// TIA Portal project "Dual_Transport_Line" (V19)

(* hardware
DEVICE "S7-1200 station_1"  S7-1200 Station
   slot 0: "Rack_0"  S7-1200 Rack  Rack  V1.0
   slot 1: "PLC_1"  CPU 1215C AC/DC/Rly  6ES7 215-1BG40-0XB0  V4.6
DEVICE "HMI_1"  KTP400 Basic PN
   slot 0: "HMI_1"  KTP400 Basic PN  6AV2 123-2DB03-0AX0  15.1.0.0
   slot 1: "HMI_RT_1"  KTP400 Basic PN  6AV2 123-2DB03-0AX0  15.1.0.0
   slot 5: "HMI_1.IE_CP_1"  PROFINET Interface  15.0.1.0
      slot 1: "PROFINET Interface_1"  PROFINET Interface
         slot 1: "Port_1"  Port
*)

// ===== PLC "PLC_1"  CPU 1215C AC/DC/Rly =====

VAR_GLOBAL   // PLC tag table "Default tag table"
   "System_Byte" AT %MB1 : Byte;
   "FirstScan" AT %M1.0 : Bool;
   "DiagStatusUpdate" AT %M1.1 : Bool;
   "AlwaysTRUE" AT %M1.2 : Bool;
   "AlwaysFALSE" AT %M1.3 : Bool;
   "Clock_Byte" AT %MB0 : Byte;
   "Clock_10Hz" AT %M0.0 : Bool;
   "Clock_5Hz" AT %M0.1 : Bool;
   "Clock_2.5Hz" AT %M0.2 : Bool;
   "Clock_2Hz" AT %M0.3 : Bool;
   "Clock_1.25Hz" AT %M0.4 : Bool;
   "Clock_1Hz" AT %M0.5 : Bool;
   "Clock_0.625Hz" AT %M0.6 : Bool;
   "Clock_0.5Hz" AT %M0.7 : Bool;
END_VAR

VAR_GLOBAL   // PLC tag table "IO"
   "MPCB_01" AT %I0.0 : Bool;   // Motor Protection Circuit Breaker
   "MPCB_02" AT %I0.1 : Bool;   // Motor Protection Circuit Breaker
   "Motor_01" AT %Q0.0 : Bool;
   "Motor_02" AT %Q0.1 : Bool;
END_VAR

TYPE "UDT_Statehandler"
   STRUCT
      State : Struct
         xReady : Bool;
         xRunning : Bool;
         xReset : Bool;
         xFaulted : Bool;
         iState : Int;
      END_STRUCT;
      Command : Struct
         xStart : Bool;
         xStop : Bool;
         xReset : Bool;
      END_STRUCT;
   END_STRUCT;
END_TYPE

TYPE "UDT_Transporter"
   STRUCT
      Status : Struct
         xWith_Package : Bool;
         xFaulted : Bool;
         xRunning : Bool;
         iState : Int;   // 0 - Stop; 10 - Running; 20 - Faulted
      END_STRUCT;
      Command : Struct
         xStart_Sensor : Bool;
         xEnd_Sensor : Bool;
      END_STRUCT;
      Configuration : Struct
         tDowntime : Int;
         iSpeed : Int;
      END_STRUCT;
      Faulted : Struct
         wTrigger : Word;
      END_STRUCT;
   END_STRUCT;
END_TYPE

DATA_BLOCK "Instance - FB - Mirror"   // DB7
{ S7_Optimized_Access := 'TRUE' }
VERSION : 0.1
// stored: InstanceOfName FB - Mirror
"FB - Mirror"
BEGIN
END_DATA_BLOCK

// folder: 00 Machine

DATA_BLOCK "Instance - FB - Statehandler"   // DB2
{ S7_Optimized_Access := 'TRUE' }
VERSION : 0.1
// stored: InstanceOfName FB - Statehandler
"FB - Statehandler"
BEGIN
END_DATA_BLOCK

DATA_BLOCK "Instance - FB - Machine Modules"   // DB3
{ S7_Optimized_Access := 'TRUE' }
VERSION : 0.1
// stored: InstanceOfName FB - Machine Modules
"FB - Machine Modules"
BEGIN
END_DATA_BLOCK

// folder: 01 Equipment/01 Instance

DATA_BLOCK "Instance - FB - Transporter_02"   // DB4
{ S7_Optimized_Access := 'TRUE' }
VERSION : 0.1
// stored: InstanceOfName FB - Transporter
"FB - Transporter"
BEGIN
END_DATA_BLOCK

DATA_BLOCK "Instance - FB - Transporter_01"   // DB6
{ S7_Optimized_Access := 'TRUE' }
VERSION : 0.1
// stored: InstanceOfName FB - Transporter
"FB - Transporter"
BEGIN
END_DATA_BLOCK

DATA_BLOCK "Instance - FB - Equipment Modules"   // DB8
{ S7_Optimized_Access := 'TRUE' }
VERSION : 0.1
// stored: InstanceOfName FB - Equipment Module
"FB - Equipment Module"
BEGIN
END_DATA_BLOCK

DATA_BLOCK "Instance - FB - Package_Position"   // DB9
{ S7_Optimized_Access := 'TRUE' }
VERSION : 0.1
// stored: InstanceOfName FB - Package_Position
"FB - Package_Position"
BEGIN
END_DATA_BLOCK

DATA_BLOCK "Instance - FB - Sensor_01"   // DB10
{ S7_Optimized_Access := 'TRUE' }
VERSION : 0.1
// stored: InstanceOfName FB - Sensor
"FB - Sensor"
BEGIN
END_DATA_BLOCK

DATA_BLOCK "Instance - FB - Sensor_02"   // DB11
{ S7_Optimized_Access := 'TRUE' }
VERSION : 0.1
// stored: InstanceOfName FB - Sensor
"FB - Sensor"
BEGIN
END_DATA_BLOCK

DATA_BLOCK "Instance - Package_Counter"   // DB12
{ S7_Optimized_Access := 'TRUE' }
VERSION : 0.1
// stored: InstanceOfName Package_Counter
"Package_Counter"
BEGIN
END_DATA_BLOCK

// folder: 02 Global Data

DATA_BLOCK "DB - Statehandler"   // DB1
{ S7_Optimized_Access := 'TRUE' }
VERSION : 0.1
   VAR
      Statehandler : "UDT_Statehandler";
   END_VAR
BEGIN
END_DATA_BLOCK

DATA_BLOCK "DB - Equipment"   // DB5
{ S7_Optimized_Access := 'TRUE' }
VERSION : 0.1
   VAR
      Transporter_01 : "UDT_Transporter";
      Transporter_02 : "UDT_Transporter";
      iPackage_Position : Int;
      iPackage_Count : Int;
   END_VAR
BEGIN
END_DATA_BLOCK

// folder: (top level)

FUNCTION_BLOCK "FB - Mirror"   // FB3, LAD
{ S7_Optimized_Access := 'TRUE' }
VERSION : 0.1
BEGIN

REGION Network 1: Motor Protection Circuit Breaker
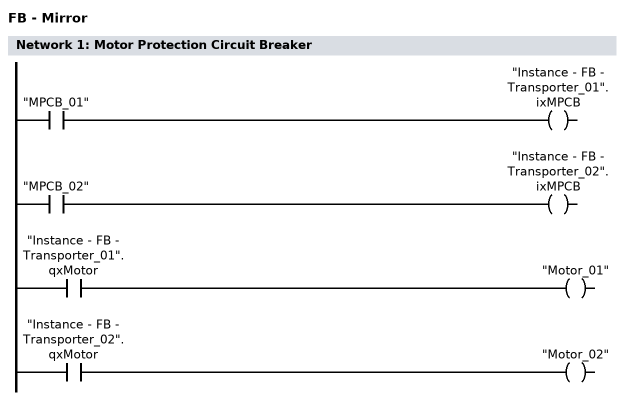
   RUNG wire#powerrail
      Contact( "MPCB_01" )
      Coil( "Instance - FB - Transporter_01".ixMPCB )
   END_RUNG
   RUNG wire#powerrail
      Contact( "MPCB_02" )
      Coil( "Instance - FB - Transporter_02".ixMPCB )
   END_RUNG
   RUNG wire#powerrail
      Contact( "Instance - FB - Transporter_01".qxMotor )
      Coil( "Motor_01" )
   END_RUNG
   RUNG wire#powerrail
      Contact( "Instance - FB - Transporter_02".qxMotor )
      Coil( "Motor_02" )
   END_RUNG
   // the same network as SCL:
   "Instance - FB - Transporter_01".ixMPCB := "MPCB_01";
   "Instance - FB - Transporter_02".ixMPCB := "MPCB_02";
   "Motor_01" := "Instance - FB - Transporter_01".qxMotor;
   "Motor_02" := "Instance - FB - Transporter_02".qxMotor;
END_REGION
END_FUNCTION_BLOCK

ORGANIZATION_BLOCK "Main"   // OB1, LAD, ProgramCycle
TITLE = "Main Program Sweep (Cycle)"
{ S7_Optimized_Access := 'TRUE' }
VERSION : 0.1
   VAR_INPUT
      Initial_Call : Bool;   // Initial call of this OB
      Remanence : Bool;   // =True, if remanent data are available
   END_VAR
BEGIN

REGION Network 1: CALL MACHINE MODULES
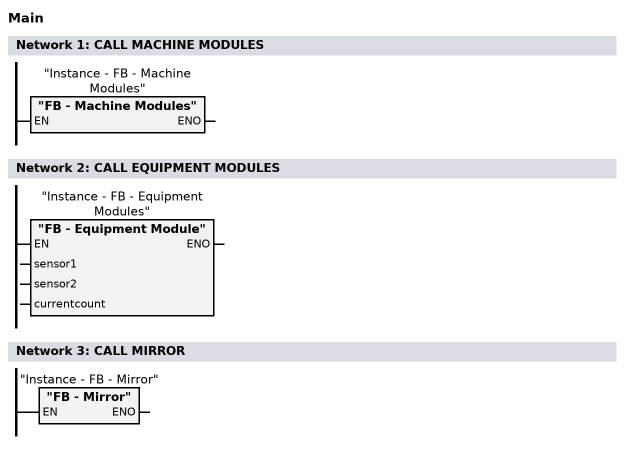
   RUNG wire#powerrail
      "Instance - FB - Machine Modules"()
   END_RUNG
   // the same network as SCL:
   "Instance - FB - Machine Modules"();   // "FB - Machine Modules"
END_REGION

REGION Network 2: CALL EQUIPMENT MODULES
   RUNG wire#powerrail
      "Instance - FB - Equipment Modules"(sensor1 :=, sensor2 :=, currentcount :=)
   END_RUNG
   // the same network as SCL:
   "Instance - FB - Equipment Modules"();   // "FB - Equipment Module"
END_REGION

REGION Network 3: CALL MIRROR
   RUNG wire#powerrail
      "Instance - FB - Mirror"()
   END_RUNG
   // the same network as SCL:
   "Instance - FB - Mirror"();   // "FB - Mirror"
END_REGION
END_ORGANIZATION_BLOCK

// folder: 00 Machine

FUNCTION_BLOCK "FB - Statehandler"   // FB1, LAD
{ S7_Optimized_Access := 'TRUE' }
VERSION : 0.1
   VAR_INPUT
      Transporter_01 : "UDT_Transporter";
      Transporter_02 : "UDT_Transporter";
   END_VAR
   VAR_IN_OUT
      "DB Statehandler" : "UDT_Statehandler";
   END_VAR
   VAR
      "xActive Faulted" : Bool;
      R_TRIG_Start : R_TRIG;
      R_TRIG_Stop : R_TRIG;
      R_TRIG_Reset : R_TRIG;
      xGlobal_Faulted : Bool;
   END_VAR
BEGIN

REGION Network 1: GLOBAL FAULTED
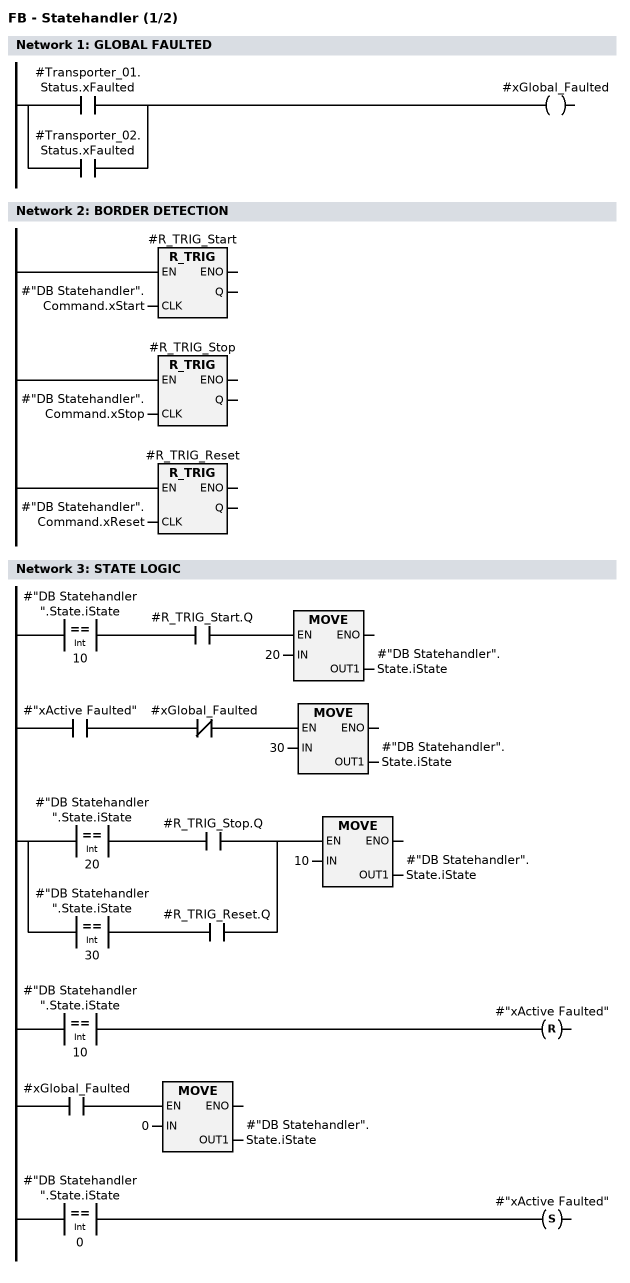
   RUNG wire#powerrail
      Contact( #Transporter_01.Status.xFaulted )
      wire#w1
      Coil( #xGlobal_Faulted )
   END_RUNG
   RUNG wire#powerrail
      Contact( #Transporter_02.Status.xFaulted )
   END_RUNG wire#w1
   // the same network as SCL:
   #xGlobal_Faulted := #Transporter_01.Status.xFaulted OR #Transporter_02.Status.xFaulted;
END_REGION

REGION Network 2: BORDER DETECTION
   #R_TRIG_Start(CLK := #"DB Statehandler".Command.xStart);   // R_TRIG
   #R_TRIG_Stop(CLK := #"DB Statehandler".Command.xStop);   // R_TRIG
   #R_TRIG_Reset(CLK := #"DB Statehandler".Command.xReset);   // R_TRIG
END_REGION

REGION Network 3: STATE LOGIC
   RUNG wire#powerrail
      { S7_Templates := "SrcType := Int" } EQ_Contact(in1 := #"DB Statehandler".State.iState, in2 := 10)
      Contact( #R_TRIG_Start.Q )
      Move(in := 20, out1 => #"DB Statehandler".State.iState)
   END_RUNG
   RUNG wire#powerrail
      Contact( #"xActive Faulted" )
      I_Contact( #xGlobal_Faulted )
      Move(in := 30, out1 => #"DB Statehandler".State.iState)
   END_RUNG
   RUNG wire#powerrail
      { S7_Templates := "SrcType := Int" } EQ_Contact(in1 := #"DB Statehandler".State.iState, in2 := 20)
      Contact( #R_TRIG_Stop.Q )
      wire#w1
      Move(in := 10, out1 => #"DB Statehandler".State.iState)
   END_RUNG
   RUNG wire#powerrail
      { S7_Templates := "SrcType := Int" } EQ_Contact(in1 := #"DB Statehandler".State.iState, in2 := 30)
      Contact( #R_TRIG_Reset.Q )
   END_RUNG wire#w1
   RUNG wire#powerrail
      { S7_Templates := "SrcType := Int" } EQ_Contact(in1 := #"DB Statehandler".State.iState, in2 := 10)
      R_Coil( #"xActive Faulted" )
   END_RUNG
   RUNG wire#powerrail
      Contact( #xGlobal_Faulted )
      Move(in := 0, out1 => #"DB Statehandler".State.iState)
   END_RUNG
   RUNG wire#powerrail
      { S7_Templates := "SrcType := Int" } EQ_Contact(in1 := #"DB Statehandler".State.iState, in2 := 0)
      S_Coil( #"xActive Faulted" )
   END_RUNG
   // the same network as SCL:
   IF (#"DB Statehandler".State.iState = 10) AND #R_TRIG_Start.Q THEN
       #"DB Statehandler".State.iState := 20;
   END_IF;
   IF #"xActive Faulted" AND NOT #xGlobal_Faulted THEN #"DB Statehandler".State.iState := 30; END_IF;
   IF ((#"DB Statehandler".State.iState = 20) AND #R_TRIG_Stop.Q) OR ((#"DB Statehandler".State.iState = 30) AND #R_TRIG_Reset.Q) THEN
       #"DB Statehandler".State.iState := 10;
   END_IF;
   IF #"DB Statehandler".State.iState = 10 THEN #"xActive Faulted" := FALSE; END_IF;
   IF #xGlobal_Faulted THEN #"DB Statehandler".State.iState := 0; END_IF;
   IF #"DB Statehandler".State.iState = 0 THEN #"xActive Faulted" := TRUE; END_IF;
END_REGION

REGION Network 4: TRIGGERS
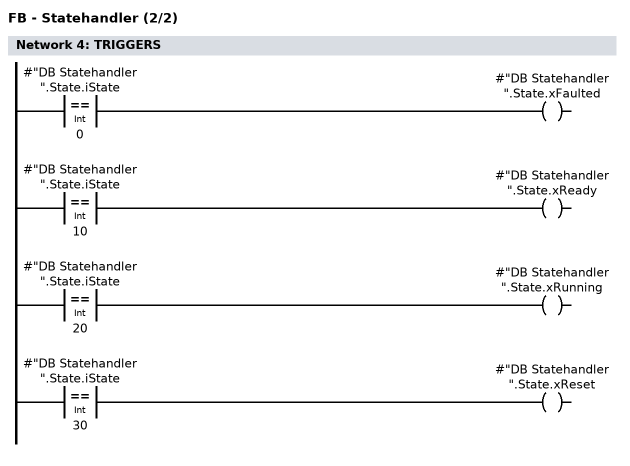
   RUNG wire#powerrail
      { S7_Templates := "SrcType := Int" } EQ_Contact(in1 := #"DB Statehandler".State.iState, in2 := 0)
      Coil( #"DB Statehandler".State.xFaulted )
   END_RUNG
   RUNG wire#powerrail
      { S7_Templates := "SrcType := Int" } EQ_Contact(in1 := #"DB Statehandler".State.iState, in2 := 10)
      Coil( #"DB Statehandler".State.xReady )
   END_RUNG
   RUNG wire#powerrail
      { S7_Templates := "SrcType := Int" } EQ_Contact(in1 := #"DB Statehandler".State.iState, in2 := 20)
      Coil( #"DB Statehandler".State.xRunning )
   END_RUNG
   RUNG wire#powerrail
      { S7_Templates := "SrcType := Int" } EQ_Contact(in1 := #"DB Statehandler".State.iState, in2 := 30)
      Coil( #"DB Statehandler".State.xReset )
   END_RUNG
   // the same network as SCL:
   #"DB Statehandler".State.xFaulted := #"DB Statehandler".State.iState = 0;
   #"DB Statehandler".State.xReady := #"DB Statehandler".State.iState = 10;
   #"DB Statehandler".State.xRunning := #"DB Statehandler".State.iState = 20;
   #"DB Statehandler".State.xReset := #"DB Statehandler".State.iState = 30;
END_REGION
END_FUNCTION_BLOCK

FUNCTION_BLOCK "FB - Machine Modules"   // FB2, LAD
{ S7_Optimized_Access := 'TRUE' }
VERSION : 0.1
BEGIN

REGION Network 1
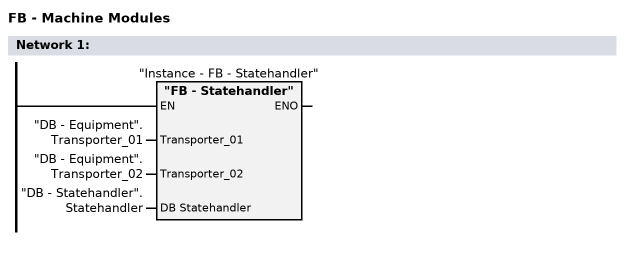
   RUNG wire#powerrail
      "Instance - FB - Statehandler"(Transporter_01 := "DB - Equipment".Transporter_01, Transporter_02 := "DB - Equipment".Transporter_02, "DB Statehandler" := "DB - Statehandler".Statehandler)
   END_RUNG
   // the same network as SCL:
   "Instance - FB - Statehandler"(Transporter_01 := "DB - Equipment".Transporter_01,   // "FB - Statehandler"
                           Transporter_02 := "DB - Equipment".Transporter_02,
                           "DB Statehandler" := "DB - Statehandler".Statehandler);
END_REGION
END_FUNCTION_BLOCK

// folder: 01 Equipment/00 Function

FUNCTION_BLOCK "FB - Equipment Module"   // FB4, LAD
{ S7_Optimized_Access := 'TRUE' }
VERSION : 0.1
   VAR_INPUT
      sensor1 : Bool;
      sensor2 : Bool;
      currentcount : DInt;
   END_VAR
BEGIN

REGION Network 1: CALL TRANSPORTER
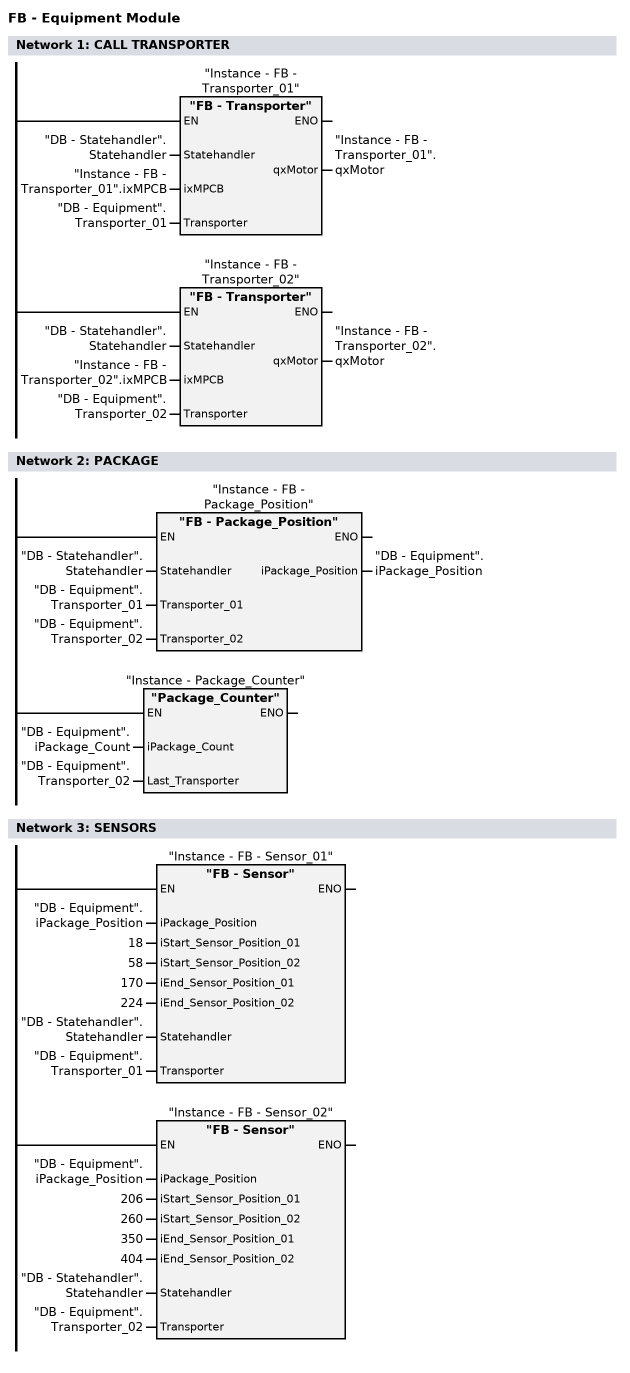
   RUNG wire#powerrail
      "Instance - FB - Transporter_01"(Statehandler := "DB - Statehandler".Statehandler, ixMPCB := "Instance - FB - Transporter_01".ixMPCB, Transporter := "DB - Equipment".Transporter_01, qxMotor => "Instance - FB - Transporter_01".qxMotor)
   END_RUNG
   RUNG wire#powerrail
      "Instance - FB - Transporter_02"(Statehandler := "DB - Statehandler".Statehandler, ixMPCB := "Instance - FB - Transporter_02".ixMPCB, Transporter := "DB - Equipment".Transporter_02, qxMotor => "Instance - FB - Transporter_02".qxMotor)
   END_RUNG
   // the same network as SCL:
   "Instance - FB - Transporter_01"(Statehandler := "DB - Statehandler".Statehandler,   // "FB - Transporter"
                           ixMPCB := "Instance - FB - Transporter_01".ixMPCB,
                           Transporter := "DB - Equipment".Transporter_01,
                           qxMotor => "Instance - FB - Transporter_01".qxMotor);
   "Instance - FB - Transporter_02"(Statehandler := "DB - Statehandler".Statehandler,   // "FB - Transporter"
                           ixMPCB := "Instance - FB - Transporter_02".ixMPCB,
                           Transporter := "DB - Equipment".Transporter_02,
                           qxMotor => "Instance - FB - Transporter_02".qxMotor);
END_REGION

REGION Network 2: PACKAGE
   RUNG wire#powerrail
      "Instance - FB - Package_Position"(Statehandler := "DB - Statehandler".Statehandler, Transporter_01 := "DB - Equipment".Transporter_01, Transporter_02 := "DB - Equipment".Transporter_02, iPackage_Position => "DB - Equipment".iPackage_Position)
   END_RUNG
   RUNG wire#powerrail
      "Instance - Package_Counter"(iPackage_Count := "DB - Equipment".iPackage_Count, Last_Transporter := "DB - Equipment".Transporter_02)
   END_RUNG
   // the same network as SCL:
   "Instance - FB - Package_Position"(Statehandler := "DB - Statehandler".Statehandler,   // "FB - Package_Position"
                           Transporter_01 := "DB - Equipment".Transporter_01,
                           Transporter_02 := "DB - Equipment".Transporter_02,
                           iPackage_Position => "DB - Equipment".iPackage_Position);
   "Instance - Package_Counter"(iPackage_Count := "DB - Equipment".iPackage_Count,   // "Package_Counter"
                           Last_Transporter := "DB - Equipment".Transporter_02);
END_REGION

REGION Network 3: SENSORS
   RUNG wire#powerrail
      "Instance - FB - Sensor_01"(iPackage_Position := "DB - Equipment".iPackage_Position, iStart_Sensor_Position_01 := 18, iStart_Sensor_Position_02 := 58, iEnd_Sensor_Position_01 := 170, iEnd_Sensor_Position_02 := 224, Statehandler := "DB - Statehandler".Statehandler, Transporter := "DB - Equipment".Transporter_01)
   END_RUNG
   RUNG wire#powerrail
      "Instance - FB - Sensor_02"(iPackage_Position := "DB - Equipment".iPackage_Position, iStart_Sensor_Position_01 := 206, iStart_Sensor_Position_02 := 260, iEnd_Sensor_Position_01 := 350, iEnd_Sensor_Position_02 := 404, Statehandler := "DB - Statehandler".Statehandler, Transporter := "DB - Equipment".Transporter_02)
   END_RUNG
   // the same network as SCL:
   "Instance - FB - Sensor_01"(iPackage_Position := "DB - Equipment".iPackage_Position,   // "FB - Sensor"
                           iStart_Sensor_Position_01 := 18,
                           iStart_Sensor_Position_02 := 58,
                           iEnd_Sensor_Position_01 := 170,
                           iEnd_Sensor_Position_02 := 224,
                           Statehandler := "DB - Statehandler".Statehandler,
                           Transporter := "DB - Equipment".Transporter_01);
   "Instance - FB - Sensor_02"(iPackage_Position := "DB - Equipment".iPackage_Position,   // "FB - Sensor"
                           iStart_Sensor_Position_01 := 206,
                           iStart_Sensor_Position_02 := 260,
                           iEnd_Sensor_Position_01 := 350,
                           iEnd_Sensor_Position_02 := 404,
                           Statehandler := "DB - Statehandler".Statehandler,
                           Transporter := "DB - Equipment".Transporter_02);
END_REGION
END_FUNCTION_BLOCK

FUNCTION_BLOCK "FB - Transporter"   // FB5, LAD
{ S7_Optimized_Access := 'TRUE' }
VERSION : 0.1
   VAR_INPUT
      Statehandler : "UDT_Statehandler";
      ixMPCB : Bool;   // Motor Protection Circuit Breaker
   END_VAR
   VAR_OUTPUT
      qxMotor : Bool;
   END_VAR
   VAR_IN_OUT
      Transporter : "UDT_Transporter";
   END_VAR
   VAR
      F_TRIG_Sensor_End : F_TRIG;
      TOF_Downtime : TOF_TIME;
      iDowntime_MS : DInt;
   END_VAR
BEGIN

REGION Network 1: CONVERT UNITS
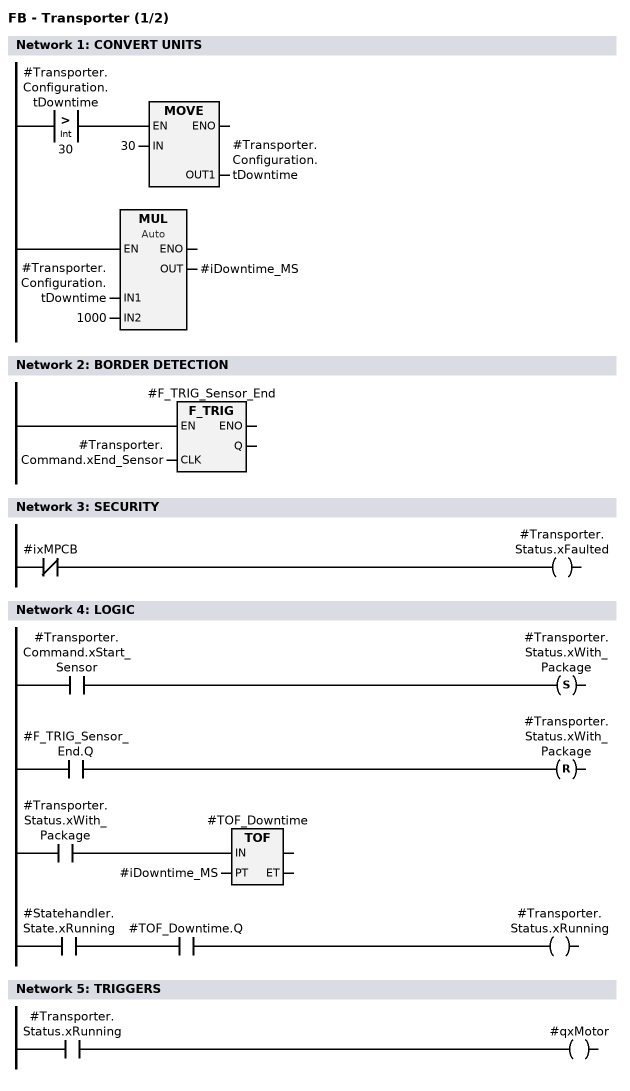
   RUNG wire#powerrail
      { S7_Templates := "SrcType := Int" } GT_Contact(in1 := #Transporter.Configuration.tDowntime, in2 := 30)
      Move(in := 30, out1 => #Transporter.Configuration.tDowntime)
   END_RUNG
   RUNG wire#powerrail
      Mul(in1 := #Transporter.Configuration.tDowntime, in2 := 1000, out => #iDowntime_MS)
   END_RUNG
   // the same network as SCL:
   IF #Transporter.Configuration.tDowntime > 30 THEN #Transporter.Configuration.tDowntime := 30; END_IF;
   #iDowntime_MS := #Transporter.Configuration.tDowntime * 1000;
END_REGION

REGION Network 2: BORDER DETECTION
   #F_TRIG_Sensor_End(CLK := #Transporter.Command.xEnd_Sensor);   // F_TRIG
END_REGION

REGION Network 3: SECURITY
   RUNG wire#powerrail
      I_Contact( #ixMPCB )
      Coil( #Transporter.Status.xFaulted )
   END_RUNG
   // the same network as SCL:
   #Transporter.Status.xFaulted := NOT #ixMPCB;
END_REGION

REGION Network 4: LOGIC
   IF #Transporter.Command.xStart_Sensor THEN #Transporter.Status.xWith_Package := TRUE; END_IF;
   IF #F_TRIG_Sensor_End.Q THEN #Transporter.Status.xWith_Package := FALSE; END_IF;
   #TOF_Downtime(IN := #Transporter.Status.xWith_Package, PT := #iDowntime_MS);   // TOF
   #Transporter.Status.xRunning := #Statehandler.State.xRunning AND #TOF_Downtime.Q;
END_REGION

REGION Network 5: TRIGGERS
   RUNG wire#powerrail
      Contact( #Transporter.Status.xRunning )
      Coil( #qxMotor )
   END_RUNG
   // the same network as SCL:
   #qxMotor := #Transporter.Status.xRunning;
END_REGION

REGION Network 6: STATUS
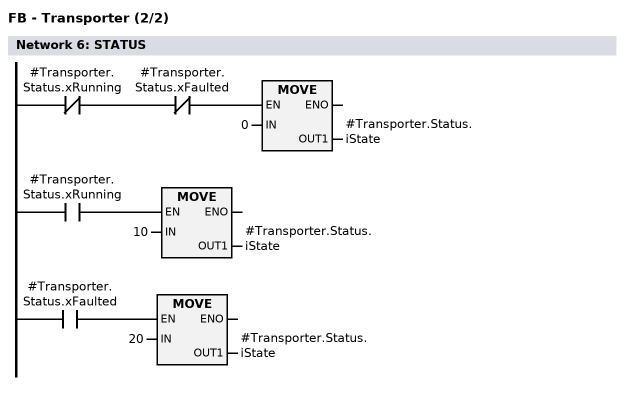
   RUNG wire#powerrail
      I_Contact( #Transporter.Status.xRunning )
      I_Contact( #Transporter.Status.xFaulted )
      Move(in := 0, out1 => #Transporter.Status.iState)
   END_RUNG
   RUNG wire#powerrail
      Contact( #Transporter.Status.xRunning )
      Move(in := 10, out1 => #Transporter.Status.iState)
   END_RUNG
   RUNG wire#powerrail
      Contact( #Transporter.Status.xFaulted )
      Move(in := 20, out1 => #Transporter.Status.iState)
   END_RUNG
   // the same network as SCL:
   IF NOT #Transporter.Status.xRunning AND NOT #Transporter.Status.xFaulted THEN
       #Transporter.Status.iState := 0;
   END_IF;
   IF #Transporter.Status.xRunning THEN #Transporter.Status.iState := 10; END_IF;
   IF #Transporter.Status.xFaulted THEN #Transporter.Status.iState := 20; END_IF;
END_REGION
END_FUNCTION_BLOCK

FUNCTION_BLOCK "FB - Package_Position"   // FB6, LAD
{ S7_Optimized_Access := 'TRUE' }
VERSION : 0.1
   VAR_OUTPUT
      iPackage_Position : Int := 36;
   END_VAR
   VAR_IN_OUT
      Statehandler : "UDT_Statehandler";
      Transporter_01 : "UDT_Transporter";
      Transporter_02 : "UDT_Transporter";
   END_VAR
   VAR
      R_TRIG_Clock : R_TRIG;
      "Instance - FB - Clock_Transporter_01" : "FB - Clock";
      "Instance - FB - Clock_Transporter_02" : "FB - Clock";
      rRPM_Norm_Transporter_02 : Real;
      iTime_Before_Convert_01 : Int;
      iTime_Before_Convert_02 : DInt;
      tTime_Transporter_01 : Time;
      tTime_Transporter_02 : Time;
   END_VAR
BEGIN

REGION Network 1: CLOCK
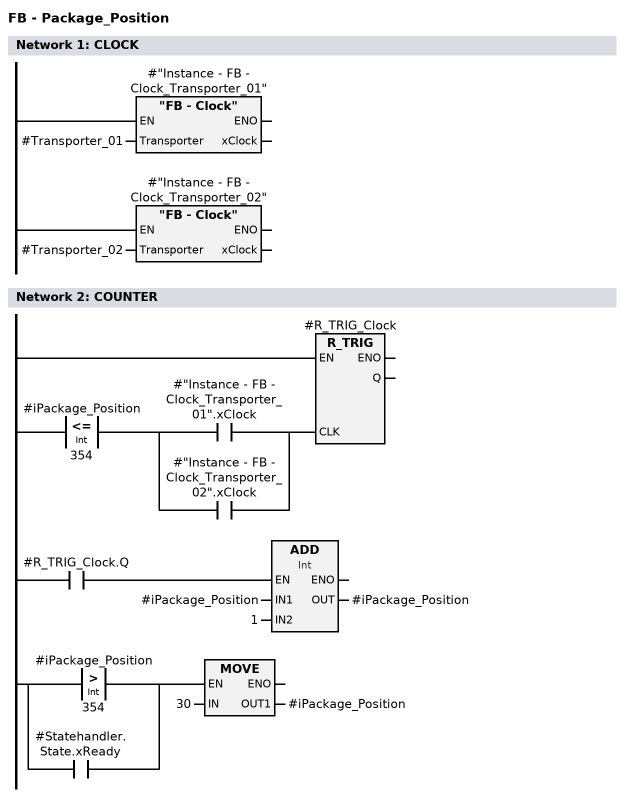
   RUNG wire#powerrail
      #"Instance - FB - Clock_Transporter_01"(Transporter := #Transporter_01, xClock =>)
   END_RUNG
   RUNG wire#powerrail
      #"Instance - FB - Clock_Transporter_02"(Transporter := #Transporter_02, xClock =>)
   END_RUNG
   // the same network as SCL:
   #"Instance - FB - Clock_Transporter_01"(Transporter := #Transporter_01);   // "FB - Clock"
   #"Instance - FB - Clock_Transporter_02"(Transporter := #Transporter_02);   // "FB - Clock"
END_REGION

REGION Network 2: COUNTER
   #R_TRIG_Clock(CLK := (#iPackage_Position <= 354) AND (#"Instance - FB - Clock_Transporter_01".xClock OR #"Instance - FB - Clock_Transporter_02".xClock));   // R_TRIG
   IF #R_TRIG_Clock.Q THEN #iPackage_Position := #iPackage_Position + 1; END_IF;
   IF (#iPackage_Position > 354) OR #Statehandler.State.xReady THEN #iPackage_Position := 30; END_IF;
END_REGION
END_FUNCTION_BLOCK

FUNCTION_BLOCK "FB - Sensor"   // FB7, LAD
{ S7_Optimized_Access := 'TRUE' }
VERSION : 0.1
   VAR_INPUT
      iPackage_Position : Int;
      iStart_Sensor_Position_01 : Int;
      iStart_Sensor_Position_02 : Int;
      iEnd_Sensor_Position_01 : Int;
      iEnd_Sensor_Position_02 : Int;
   END_VAR
   VAR_IN_OUT
      Statehandler : "UDT_Statehandler";
      Transporter : "UDT_Transporter";
   END_VAR
BEGIN

REGION Network 1
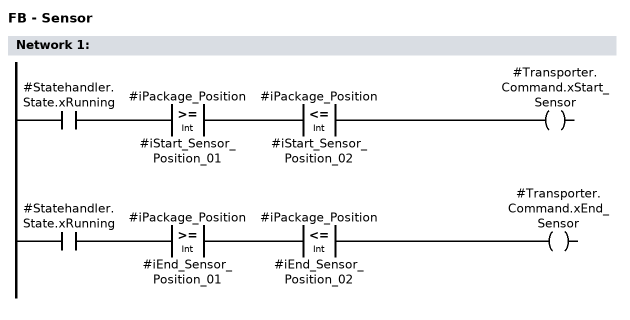
   RUNG wire#powerrail
      Contact( #Statehandler.State.xRunning )
      { S7_Templates := "SrcType := Int" } GE_Contact(in1 := #iPackage_Position, in2 := #iStart_Sensor_Position_01)
      { S7_Templates := "SrcType := Int" } LE_Contact(in1 := #iPackage_Position, in2 := #iStart_Sensor_Position_02)
      Coil( #Transporter.Command.xStart_Sensor )
   END_RUNG
   RUNG wire#powerrail
      Contact( #Statehandler.State.xRunning )
      { S7_Templates := "SrcType := Int" } GE_Contact(in1 := #iPackage_Position, in2 := #iEnd_Sensor_Position_01)
      { S7_Templates := "SrcType := Int" } LE_Contact(in1 := #iPackage_Position, in2 := #iEnd_Sensor_Position_02)
      Coil( #Transporter.Command.xEnd_Sensor )
   END_RUNG
   // the same network as SCL:
   #Transporter.Command.xStart_Sensor := #Statehandler.State.xRunning AND (#iPackage_Position >= #iStart_Sensor_Position_01) AND (#iPackage_Position <= #iStart_Sensor_Position_02);
   #Transporter.Command.xEnd_Sensor := #Statehandler.State.xRunning AND (#iPackage_Position >= #iEnd_Sensor_Position_01) AND (#iPackage_Position <= #iEnd_Sensor_Position_02);
END_REGION
END_FUNCTION_BLOCK

FUNCTION_BLOCK "Package_Counter"   // FB8, LAD
{ S7_Optimized_Access := 'TRUE' }
VERSION : 0.1
   VAR_IN_OUT
      iPackage_Count : Int;
      Last_Transporter : "UDT_Transporter";
   END_VAR
   VAR RETAIN
      "Counter" : CTU_INT;
   END_VAR
BEGIN

REGION Network 1
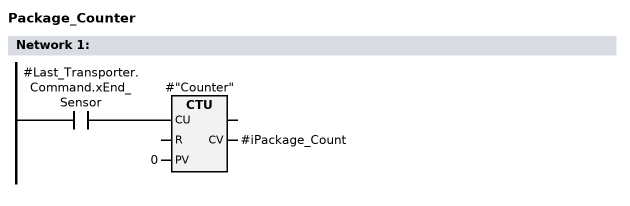
   #"Counter"(CU := #Last_Transporter.Command.xEnd_Sensor, PV := 0, CV => #iPackage_Count);   // CTU
END_REGION
END_FUNCTION_BLOCK

FUNCTION_BLOCK "FB - Clock"   // FB9, LAD
{ S7_Optimized_Access := 'TRUE' }
VERSION : 0.1
   VAR_OUTPUT
      xClock : Bool;
   END_VAR
   VAR_IN_OUT
      Transporter : "UDT_Transporter";
   END_VAR
   VAR
      TON_01 : TON_TIME;
      TON_02 : TON_TIME;
      rSpeed_Convert : Real;
      rTIme_Calculated : Real;
      iTime_Calculated : DInt;
      tTIme : Time;
   END_VAR
BEGIN

REGION Network 1: SPEED LIMIT
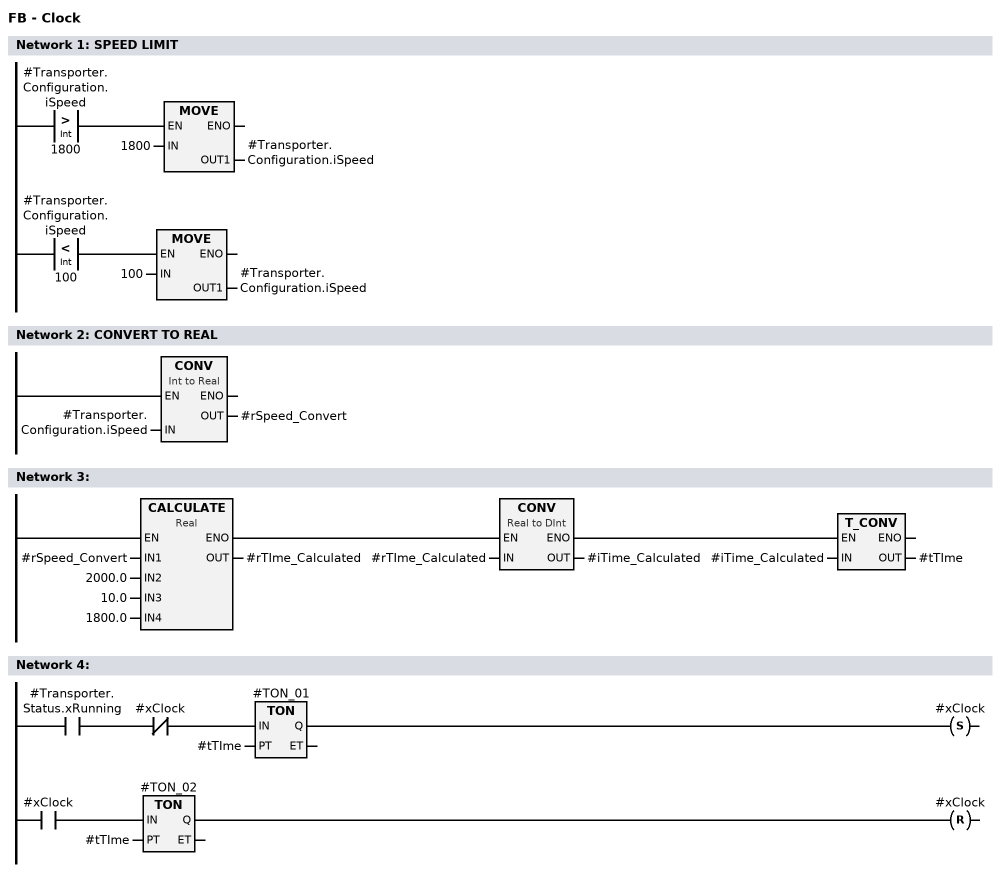
   RUNG wire#powerrail
      { S7_Templates := "SrcType := Int" } GT_Contact(in1 := #Transporter.Configuration.iSpeed, in2 := 1800)
      Move(in := 1800, out1 => #Transporter.Configuration.iSpeed)
   END_RUNG
   RUNG wire#powerrail
      { S7_Templates := "SrcType := Int" } LT_Contact(in1 := #Transporter.Configuration.iSpeed, in2 := 100)
      Move(in := 100, out1 => #Transporter.Configuration.iSpeed)
   END_RUNG
   // the same network as SCL:
   IF #Transporter.Configuration.iSpeed > 1800 THEN #Transporter.Configuration.iSpeed := 1800; END_IF;
   IF #Transporter.Configuration.iSpeed < 100 THEN #Transporter.Configuration.iSpeed := 100; END_IF;
END_REGION

REGION Network 2: CONVERT TO REAL
   RUNG wire#powerrail
      { S7_Templates := "[SrcType := Int, DestType := Real]" } Convert(in := #Transporter.Configuration.iSpeed, out => #rSpeed_Convert)
   END_RUNG
   // the same network as SCL:
   #rSpeed_Convert := INT_TO_REAL(#Transporter.Configuration.iSpeed);
END_REGION

REGION Network 3
   #rTIme_Calculated := 2000.0 - ((#rSpeed_Convert / 1800.0) * (2000.0 -  10.0));
   #iTime_Calculated := REAL_TO_DINT(#rTIme_Calculated);
   #tTIme := T_CONV(IN := #iTime_Calculated);
END_REGION

REGION Network 4
   #TON_01(IN := #Transporter.Status.xRunning AND NOT #xClock, PT := #tTIme);   // TON
   IF #TON_01.Q THEN #xClock := TRUE; END_IF;
   #TON_02(IN := #xClock, PT := #tTIme);   // TON
   IF #TON_02.Q THEN #xClock := FALSE; END_IF;
END_REGION
END_FUNCTION_BLOCK

(* ===== HMI "HMI_RT_1" =====
system functions are stored by id; their names below are inferred from use
connection "HMI_Connection_1": ETHERNET, SMART_S7_1200_OMS

HMI tags "Login Tags"
   "_iScreenNumber" : Int, internal
   "_iUsername_Group" : Int, internal
   "_sUsername" : WString[254], internal
   "_sInputUsername" : WString[254], internal
   "_sInputPassword" : WString[254], internal

HMI tags "Template Command Tags"
   "_xState_Btn_Alarm" : Bool, internal
   "_xState_Btn_Overview" : Bool, internal
   "_xState_Btn_Recipes" : Bool, internal
   "_xState_Btn_Settings" : Bool, internal

HMI tags "Configuration Tags"
   "DB - Equipment_Transporter_01_Configuration_iSpeed" : Int = PLC "DB - Equipment".Transporter_01.Configuration.iSpeed, 100 ms
   "DB - Equipment_Transporter_01_Configuration_tDowntime" : Int = PLC "DB - Equipment".Transporter_01.Configuration.tDowntime, 100 ms
   "DB - Equipment_Transporter_02_Configuration_iSpeed" : Int = PLC "DB - Equipment".Transporter_02.Configuration.iSpeed, 100 ms
   "DB - Equipment_Transporter_02_Configuration_tDowntime" : Int = PLC "DB - Equipment".Transporter_02.Configuration.tDowntime, 100 ms

HMI tags "Status Tags"
   "DB - Equipment_iPackage_Count" : Int = PLC "DB - Equipment".iPackage_Count, 100 ms
   "DB - Equipment_iPackage_Position" : Int = PLC "DB - Equipment".iPackage_Position, 100 ms
   "DB - Equipment_Transporter_01_Faulted_wTrigger" : Word = PLC "DB - Equipment".Transporter_01.Faulted.wTrigger, 1 s
   "DB - Equipment_Transporter_01_Status_iState" : Int = PLC "DB - Equipment".Transporter_01.Status.iState, 100 ms
   "DB - Equipment_Transporter_02_Faulted_wTrigger" : Word = PLC "DB - Equipment".Transporter_02.Faulted.wTrigger, 1 s
   "DB - Equipment_Transporter_02_Status_iState" : Int = PLC "DB - Equipment".Transporter_02.Status.iState, 100 ms
   "DB - Statehandler_Statehandler" : UDT_Statehandler = PLC "DB - Statehandler".Statehandler AT %DB1.DBX0.0, 100 ms

analog alarms
   1: 'Fault detected in Transporter 01', class Errors, trigger "DB - Equipment_Transporter_01_Status_iState"
   2: 'Fault detected in Transporter 02', class Errors, trigger "DB - Equipment_Transporter_02_Status_iState"

graphic list "GraphicList_Btn_template_Overview": 0 'Btn_Template_Overview_Off'; 1 'Btn_Template_Overview_On'

graphic list "GraphicList_Btn_template_Alarm": 0 'Btn_Template_Alert_Off'; 1 'Btn_Template_Alert_On'

graphic list "GraphicList_Btn_template_Recipes": 0 'Btn_Template_Recipe_Off'; 1 'Btn_Template_Recipe_On'

graphic list "GraphicList_Btn_template_Settings": 0 'Btn_Template_Settings_Off'; 1 'Btn_Template_Settings_On'

graphic list "GraphicList_Motor_01": 0 'Graphic_7'; 10 'Graphic_8'; 20 'Graphic_9'

recipe "Product A": Speed_Motor_01 <- "DB - Equipment_Transporter_01_Configuration_iSpeed", Speed_Motor_02 <- "DB - Equipment_Transporter_02_Configuration_iSpeed", Downtime_Motor_01 <- "DB - Equipment_Transporter_01_Configuration_tDowntime", Downtime_Motor_02 <- "DB - Equipment_Transporter_02_Configuration_tDowntime"

Template "Template" 480x272
   Rectangle "Template_Rectangle_4" at 4,24 size 427x242
      Appearance <- "iState"
   Button "Template_Button_1" at 435,0 size 45x45; TextOff 'Text'; PictureList "GraphicList_Btn_template_Overview"
      ProcessValue <- "_xState_Btn_Overview"
      on Release: ActivateScreen("1 OVERVIEW", 0)
   Button "Template_Button_2" at 435,44 size 45x45; TextOff 'Text'; PictureList "GraphicList_Btn_template_Alarm"; Authorization "Producao"
      on Release: ActivateScreen("5 ALARMS", 0)
      ProcessValue <- "_xState_Btn_Alarm"
   Button "Template_Button_3" at 435,88 size 45x45; TextOff 'Text'; PictureList "GraphicList_Btn_template_Recipes"; Authorization "Producao"
      on Release: ActivateScreen("10 RECIPES", 0)
      ProcessValue <- "_xState_Btn_Recipes"
   Button "Template_Button_4" at 435,132 size 45x45; TextOff 'Text'; PictureList "GraphicList_Btn_template_Settings"
      on Release: ActivateScreen("20 SETTINGS", 0)
      ProcessValue <- "_xState_Btn_Settings"
   Button "Template_Button_5" at 435,227 size 45x45; TextOff 'Text'; PictureList "GraphicList_Btn_template_Overview"; PictureOff "Btn_Template_Stop_Off"; PictureOn "Btn_Template_Stop_On"; Authorization "Producao"
      ProcessValue <- "_xState_Btn_Overview"
      on Press: function_b14e0dd5("xStop", 0)
   Button "Template_Button_6" at 435,183 size 45x45; TextOff 'Text'; PictureList "GraphicList_Btn_template_Overview"; PictureOff "Btn_Template_Start_Off"; PictureOn "Btn_Template_Start_On"; Authorization "Producao"
      ProcessValue <- "_xState_Btn_Overview"
      on Press: function_b14e0dd5("xStart", 0)
   TextField "Template_Text field_3" at 204,1 size 49x18; Text 'RECIPE'
   DateTimeField "Template_Date/time field_1" at 279,1 size 145x18
   SymbolicIOField "Template_Symbolic I/O field_1" at 72,2 size 105x17; TextOff '0'; TextOn '1'; TextList "TextList_ScreenNames"
      ProcessValue <- "_iScreenNumber"
   IOField "Template_I/O field_1" at 0,2 size 62x17; FormatPattern ?????
      ProcessValue <- "_sUsername"
      Appearance <- "_iUsername_Group"

screen "1 OVERVIEW" 480x272, template "Template"
   on GenerateScreen: SetBit("_xState_Btn_Overview"); SetTag("_iScreenNumber", 1)
   on ClearScreen: ResetBit("_xState_Btn_Overview")
   Circle "Circle_2" at 390,69 size 14x14
      Appearance <- "DB - Equipment_iPackage_Position"
   Circle "Circle_4" at 246,69 size 14x14
      Appearance <- "DB - Equipment_iPackage_Position"
   Circle "Circle_1" at 210,70 size 14x14
      Appearance <- "DB - Equipment_iPackage_Position"
   Circle "Circle_3" at 58,70 size 14x14
      Appearance <- "DB - Equipment_iPackage_Position"
   TextField "HmiScreenItemData" at 16,32 size 141x22; Text 'CURRENT COUNT:'
   IOField "I/O field_1" at 160,32 size 45x22; FormatPattern 999
      ProcessValue <- "DB - Equipment_iPackage_Count"
   GraphicView "Graphic view_2" at 4,88 size 234x49; Picture "Graphic_1"
   GraphicView "Graphic view_1" at 190,88 size 234x49; Picture "Graphic_1"
   GraphicView "Graphic view_3" at 30,76 size 40x40; Picture "Graphic_2"
      HorizontalMovement <- "DB - Equipment_iPackage_Position"
   GraphicIOField "Graphic I/O field_1" at 16,143 size 71x44; PictureList "GraphicList_Motor_01"
      ProcessValue <- "DB - Equipment_Transporter_01_Status_iState"
   TextField "HmiScreenItemData_1" at 93,154 size 72x22; Text 'M - 1001'
   GraphicIOField "Graphic I/O field_2" at 223,143 size 71x44; PictureList "GraphicList_Motor_01"
      ProcessValue <- "DB - Equipment_Transporter_02_Status_iState"
   TextField "HmiScreenItemData_2" at 300,154 size 72x22; Text 'M - 1002'
   TextField "HmiScreenItemData_3" at 16,202 size 77x18; Text 'DOWNTIME:'
   IOField "I/O field_2" at 122,200 size 75x22; Authorization "Producao"; FormatPattern 99; Unit  S
      ProcessValue <- "DB - Equipment_Transporter_01_Configuration_tDowntime"
   TextField "HmiScreenItemData_4" at 16,233 size 97x18; Text 'MOTOR SPEED:'
   IOField "I/O field_3" at 122,231 size 75x22; Authorization "Producao"; FormatPattern 9999; Unit  RPM
      ProcessValue <- "DB - Equipment_Transporter_01_Configuration_iSpeed"
   TextField "HmiScreenItemData_5" at 223,202 size 77x18; Text 'DOWNTIME:'
   IOField "I/O field_4" at 332,200 size 75x22; Authorization "Producao"; FormatPattern 99; Unit  S
      ProcessValue <- "DB - Equipment_Transporter_02_Configuration_tDowntime"
   TextField "HmiScreenItemData_6" at 223,233 size 97x18; Text 'MOTOR SPEED:'
   IOField "I/O field_5" at 332,231 size 75x22; Authorization "Producao"; FormatPattern 9999; Unit  RPM
      ProcessValue <- "DB - Equipment_Transporter_02_Configuration_iSpeed"

screen "5 ALARMS" 480x272, template "Template"
   on GenerateScreen: SetBit("_xState_Btn_Alarm"); SetTag("_iScreenNumber", 5)
   on ClearScreen: ResetBit("_xState_Btn_Alarm")
   Button "Button_2" at 380,82 size 48x48; TextOff 'Text'; PictureOff "Btn_Template_AlarmHistory_Off"; PictureOn "Btn_Template_AlarmHistory_On"
      on Release: ActivateScreen("6 ALARMS HISTORY", 0)
   Button "Button_1" at 380,28 size 48x48; TextOff 'Text'; PictureOff "Btn_Template_Reset_Off"; PictureOn "Btn_Template_Reset_On"
      on Press: function_b14e0dd5("xReset", 0); function_d9204949("Alarm view_1")
   AlarmView "Alarm view_1" at 4,24 size 373x242

screen "20 SETTINGS" 480x272, template "Template"
   on GenerateScreen: SetBit("_xState_Btn_Settings"); SetTag("_iScreenNumber", 20)
   on ClearScreen: ResetBit("_xState_Btn_Settings")
   Button "Button_2" at 308,176 size 60x60; TextOff 'Text'; PictureOff "Btn_Template_Logoff_Off"; PictureOn "Btn_Template_Logoff_On"
      on Release: function_f23ef4c9()
   Button "Button_1" at 308,107 size 60x60; TextOff 'Text'; PictureOff "Btn_Template_Login_Off"; PictureOn "Btn_Template_Login_On"
      on Release: function_a9b89908("_sInputPassword", "_sInputUsername")
   TextField "Text field_2" at 225,51 size 47x17; Text 'GROUP:'
   IOField "I/O field_4" at 276,51 size 21x17; FormatPattern 99
      ProcessValue <- "_iUsername_Group"
   IOField "I/O field_1" at 50,51 size 62x17; FormatPattern ?????
      ProcessValue <- "_sUsername"
   TextField "Text field_1" at 14,51 size 37x17; Text 'USER:'
   IOField "I/O field_2" at 80,116 size 217x42; FormatPattern ????????????????????
      ProcessValue <- "_sInputUsername"
   IOField "I/O field_3" at 80,185 size 217x42; FormatPattern ????????????????????
      ProcessValue <- "_sInputPassword"

screen "10 RECIPES" 480x272, template "Template"
   on GenerateScreen: SetBit("_xState_Btn_Recipes"); SetTag("_iScreenNumber", 10)
   on ClearScreen: ResetBit("_xState_Btn_Recipes")
   RecipeView "Recipe view_1" at 4,26 size 428x238; Authorization "Producao"

screen "6 ALARMS HISTORY" 480x272, template "Template"
   on GenerateScreen: SetTag("_iScreenNumber", 6)
   AlarmView "Alarm view_1" at 4,24 size 373x242
   Button "Button_1" at 380,28 size 48x48; TextOff 'Text'; PictureOff "Btn_Template_Clear_Off"; PictureOn "Btn_Template_Clear_On"
      on Release: function_e14cd482(0)

scheduled task "Get_User_Info"
   on Action: function_f41c6f6c("_sUsername"); function_e1ab61de("_iUsername_Group")
*)